// TIA Portal V17 export
// export: Created 2024-08-09T12:52:06.4857421Z, ExportSetting WithDefaults, DisplayName Totally Integrated Automation Portal, DisplayVersion V17 Update 7, DisplayName TIA Portal Openness, DisplayVersion V17 Update 7, DisplayName TIA Portal Version Control Interface, DisplayVersion V17, DisplayName STEP 7 Professional, DisplayVersion V17 Update 7, DisplayName STEP 7 Safety, DisplayVersion V17 Update 6, DisplayName WinCC Professional, DisplayVersion V17 Update 7
DATA_BLOCK "DB_PTSUIV_TOUR"   // DB42
VERSION : 0.1
// stored: AutoNumber true, DBAccessibleFromOPCUA true, DBAccessibleFromWebserver true, IsOnlyStoredInLoadMemory false, IsWriteProtectedInAS false
   STRUCT
      DB_PTSUIV_TOUR : Array[0..4] of "S_MODULE_SUIVI_COMMUNCHARG";
   END_STRUCT;
BEGIN
END_DATA_BLOCK
